// TIA Portal V17 export
// export: Created 2025-06-26T07:49:41.4466259Z, ExportSetting WithDefaults, DisplayName Totally Integrated Automation Portal, DisplayVersion V17 Update 8, DisplayName TIA Portal Openness, DisplayVersion V17 Update 8, DisplayName TIA Portal Version Control Interface, DisplayVersion V17, DisplayName STEP 7 Professional, DisplayVersion V17 Update 8, DisplayName STEP 7 Safety, DisplayVersion V17 Update 6, DisplayName WinCC Advanced, DisplayVersion V17 Update 8
FUNCTION "State6_Running" : Void   // FC56, FBD
{ S7_Optimized_Access := 'TRUE' }
VERSION : 0.1
// stored: AutoNumber true, IsIECCheckEnabled false, SetENOAutomatically false, UDAEnableTagReadback false
   VAR_INPUT
      Active : Bool;
   END_VAR
   VAR_OUTPUT
      Stop : Bool;
      Standby : Bool;
   END_VAR
BEGIN

REGION Network 1: State number
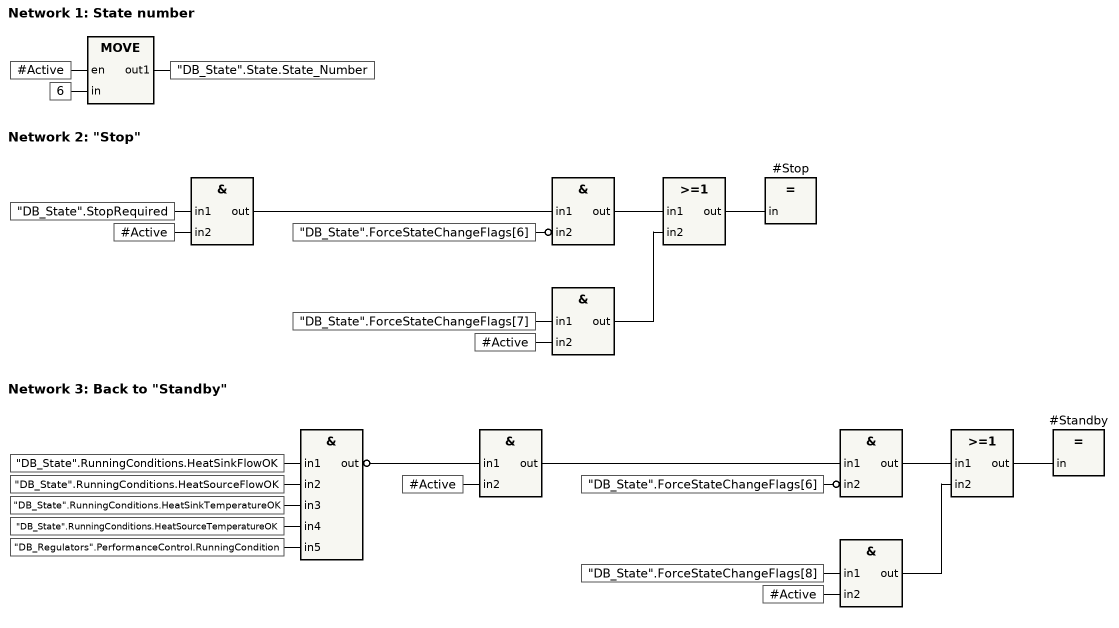
   IF #Active THEN "DB_State".State.State_Number := 6; END_IF;
END_REGION

REGION Network 2: "Stop"
   #Stop := ("DB_State".StopRequired AND #Active AND NOT "DB_State".ForceStateChangeFlags[6]) OR ("DB_State".ForceStateChangeFlags[7] AND #Active);
END_REGION

REGION Network 3: Back to "Standby"
   #Standby := (NOT ("DB_State".RunningConditions.HeatSinkFlowOK AND "DB_State".RunningConditions.HeatSourceFlowOK AND "DB_State".RunningConditions.HeatSinkTemperatureOK AND "DB_State".RunningConditions.HeatSourceTemperatureOK AND "DB_Regulators".PerformanceControl.RunningCondition) AND #Active AND NOT "DB_State".ForceStateChangeFlags[6]) OR ("DB_State".ForceStateChangeFlags[8] AND #Active);
END_REGION
END_FUNCTION
